{attribute 'GeneratedUsingTerminal: EL3483-0000-0016'}
{attribute addProperty BoxType "EL3483-0000-0016"}
{attribute addProperty Id "EtcSlaveTerminalBaseL1_StatusAT %I*L1_Status_12B1E6BB5L2_StatusAT %I*L2_Status_12B1E6BB5L3_StatusAT %I*L3_Status_12B1E6BB5Total_StatusAT %I*Total_Status_AD43C3B912Total_AdvancedAT %I*Total_Advanced_3B87F4672WcStateAT %I*WcState_9091E0EB2InfoDataAT %I*InfoData_32EB74EA10"}
{attribute addProperty CRC "3151692526"}
{attribute addProperty Size "41"}
TYPE EL3483_BBDB02EE EXTENDS EtcSlaveTerminalBase :
STRUCT
	{attribute addProperty Name "L1_Status"}
	L1_Status : L1_Status_12B1E6BB;
	{attribute addProperty Name "L2_Status"}
	L2_Status : L2_Status_12B1E6BB;
	{attribute addProperty Name "L3_Status"}
	L3_Status : L3_Status_12B1E6BB;
	{attribute addProperty Name "Total_Status"}
	Total_Status : Total_Status_AD43C3B9;
	{attribute addProperty Name "Total_Advanced"}
	Total_Advanced : Total_Advanced_3B87F467;
	{attribute addProperty Name "WcState"}
	WcState : WcState_9091E0EB;
	{attribute addProperty Name "InfoData"}
	InfoData : InfoData_32EB74EA;
END_STRUCT
END_TYPE

(* stored: Version 1.2.0.0, ProductVersion 3.1.4024.9
   DUT EL3483_BBDB02EE: Id {1bc7248d-7cd3-46dd-a5d2-f43fdaa7ae4b} *)
